Yaskawa INFORM job: 180.JBI

/JOB
//NAME 180
///FOLDERNAME INNE
//POS
///NPOS 0,0,1,0,0,0
///TOOL 0
///POSTYPE PULSE
///PULSE
EC00000=1596314,2
//INST
///DATE 2023/10/04 15:13
///ATTR SC,RW,RJ
////FRAME ROBOT
///GROUP1 ST1
NOP
MOVJ EC00000 VJ=0.78 PL=0
END
